// TIA Portal V16 export
// export: Created 2020-12-17T10:43:58.9405852Z, ExportSetting WithDefaults, WithReadOnly, DisplayName Totally Integrated Automation Portal, DisplayVersion V16 Update 2, DisplayName TIA Portal Version Control Interface, DisplayVersion V16 Update 2, DisplayName TIA Portal Openness, DisplayVersion V16 Update 2, DisplayName STEP 7 Professional, DisplayVersion V16 Update 2, DisplayName STEP 7 Safety, DisplayVersion V16, DisplayName WinCC Advanced / Unified PC, DisplayVersion V16 Update 2
TYPE "Point"
// stored: CreationDate 2020-12-17T10:41:14.5497731Z, InterfaceModifiedDate 2020-12-17T10:41:40.9176599Z, IsConsistent true, IsFailsafeCompliant false, IsKnowHowProtected false, LibraryConformanceStatus The object is library-conformant., ModifiedDate 2020-12-17T10:41:54.4302381Z
   STRUCT
      x { S7_SetPoint := 'True'} : Int := 100;
      y { S7_SetPoint := 'True'} : Int := 100;
   END_STRUCT;
END_TYPE
